Fanuc KAREL source: KF00094.KL

PROGRAM KF00094
%NOLOCKGROUP
VAR
  I: INTEGER
  J: INTEGER
  X: REAL
  Y: REAL
  B: BOOLEAN
  C: BOOLEAN
  TXT: STRING[80]
  TXT2: STRING[80]
  AI: ARRAY[4] OF INTEGER
  BI: ARRAY[4] OF INTEGER
  P: XYZWPR
  JP: JOINTPOS
  PF: POSITION
  V1: VECTOR
  V2: VECTOR
  STATUS: INTEGER
BEGIN
  V1.X = 1.0
  V2.Y = 2.0
  V1 = V1 + V2
END KF00094
